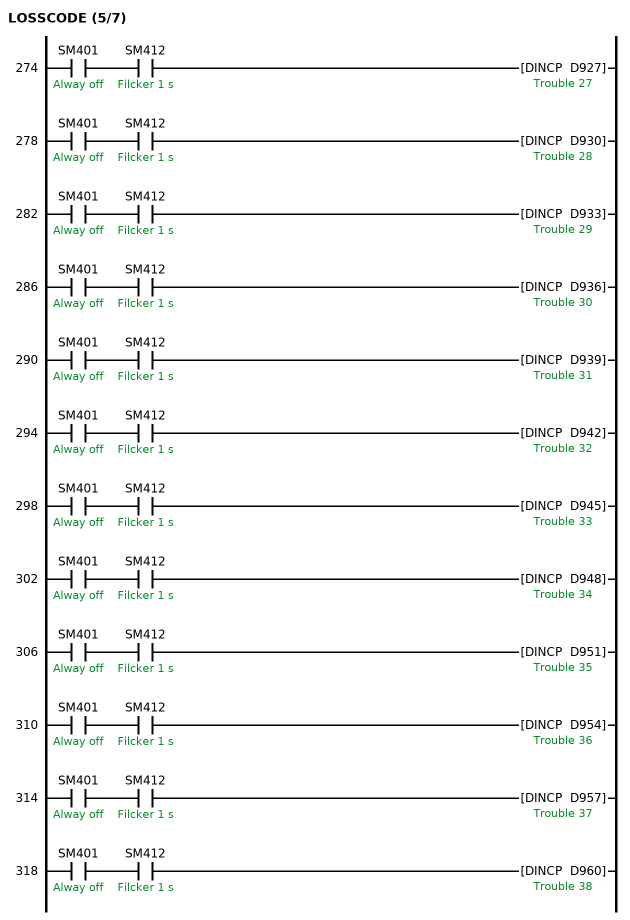
[picture p72: ladder of LOSSCODE, rungs at steps 274 to 318]
274   LD      SM401  ; Alway off
      AND     SM412  ; Filcker 1 s
      DINCP   D927  ; Trouble 27
278   LD      SM401  ; Alway off
      AND     SM412  ; Filcker 1 s
      DINCP   D930  ; Trouble 28
282   LD      SM401  ; Alway off
      AND     SM412  ; Filcker 1 s
      DINCP   D933  ; Trouble 29
286   LD      SM401  ; Alway off
      AND     SM412  ; Filcker 1 s
      DINCP   D936  ; Trouble 30
290   LD      SM401  ; Alway off
      AND     SM412  ; Filcker 1 s
      DINCP   D939  ; Trouble 31
294   LD      SM401  ; Alway off
      AND     SM412  ; Filcker 1 s
      DINCP   D942  ; Trouble 32
298   LD      SM401  ; Alway off
      AND     SM412  ; Filcker 1 s
      DINCP   D945  ; Trouble 33
302   LD      SM401  ; Alway off
      AND     SM412  ; Filcker 1 s
      DINCP   D948  ; Trouble 34
306   LD      SM401  ; Alway off
      AND     SM412  ; Filcker 1 s
      DINCP   D951  ; Trouble 35
310   LD      SM401  ; Alway off
      AND     SM412  ; Filcker 1 s
      DINCP   D954  ; Trouble 36
314   LD      SM401  ; Alway off
      AND     SM412  ; Filcker 1 s
      DINCP   D957  ; Trouble 37
318   LD      SM401  ; Alway off
      AND     SM412  ; Filcker 1 s
      DINCP   D960  ; Trouble 38
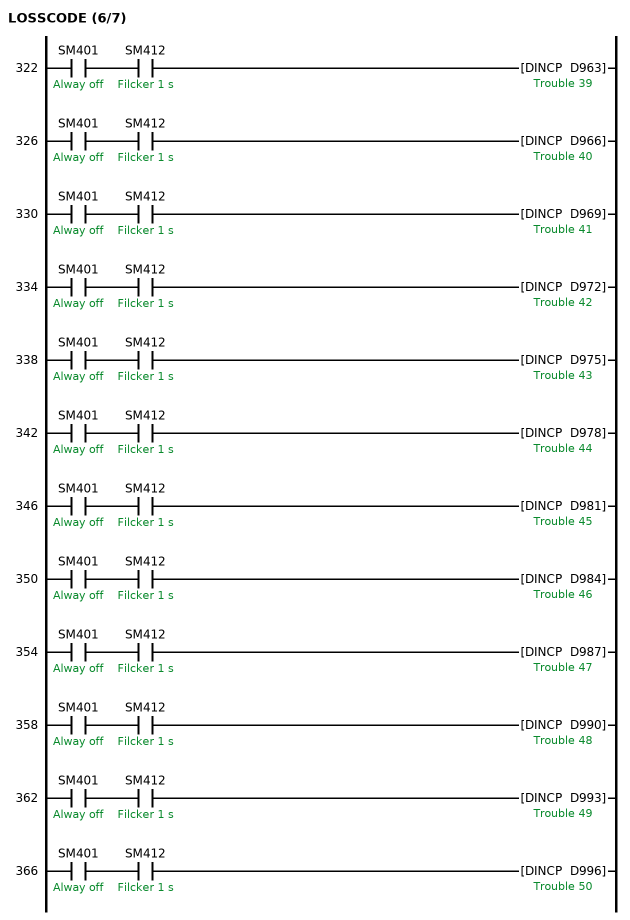
322   LD      SM401  ; Alway off
      AND     SM412  ; Filcker 1 s
      DINCP   D963  ; Trouble 39
326   LD      SM401  ; Alway off
      AND     SM412  ; Filcker 1 s
      DINCP   D966  ; Trouble 40
330   LD      SM401  ; Alway off
      AND     SM412  ; Filcker 1 s
      DINCP   D969  ; Trouble 41
334   LD      SM401  ; Alway off
      AND     SM412  ; Filcker 1 s
      DINCP   D972  ; Trouble 42
338   LD      SM401  ; Alway off
      AND     SM412  ; Filcker 1 s
      DINCP   D975  ; Trouble 43
342   LD      SM401  ; Alway off
      AND     SM412  ; Filcker 1 s
      DINCP   D978  ; Trouble 44
346   LD      SM401  ; Alway off
      AND     SM412  ; Filcker 1 s
      DINCP   D981  ; Trouble 45
350   LD      SM401  ; Alway off
      AND     SM412  ; Filcker 1 s
      DINCP   D984  ; Trouble 46
354   LD      SM401  ; Alway off
      AND     SM412  ; Filcker 1 s
      DINCP   D987  ; Trouble 47
358   LD      SM401  ; Alway off
      AND     SM412  ; Filcker 1 s
      DINCP   D990  ; Trouble 48
362   LD      SM401  ; Alway off
      AND     SM412  ; Filcker 1 s
      DINCP   D993  ; Trouble 49
366   LD      SM401  ; Alway off
      AND     SM412  ; Filcker 1 s
      DINCP   D996  ; Trouble 50
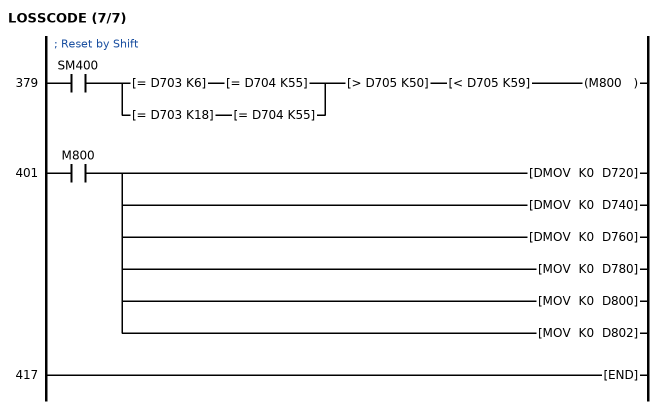
; Reset by Shift
379   LD      SM400
      LD=     D703 K6
      AND=    D704 K55
      LD=     D703 K18
      AND=    D704 K55
      ORB
      ANB
      AND>    D705 K50
      AND<    D705 K59
      OUT     M800
401   LD      M800
      DMOV    K0 D720
      DMOV    K0 D740
      DMOV    K0 D760
      MOV     K0 D780
      MOV     K0 D800
      MOV     K0 D802
417   END
END_PROGRAM
